PROGRAM PLC_Mode
VAR
END_VAR



PRG_CreateTable();

PRG_DeleteRowDatabase();

PRG_WriteDatabase();

PRG_ReadDatabase();

END_PROGRAM

(* stored: Version 1.1.0.1, ProductVersion 3.1.4024.12
   POU PLC_Mode: Id {97bd568f-b367-4734-9215-468bdf0bc17d}, SpecialFunc None *)
